{region '#Template'}
	{attribute 'Version' := '0.0.1.0'}
	{attribute 'Tags' := '"LCID": "1031", "Text": "Universal, Analog, Aggregate"'}
	{attribute 'Tags' := '"LCID": "1033", "Text": "Universal, Analog, Aggregate"'}
	{attribute 'Description' := '"LCID": "1031", "Text": "Aktor binär"'}
	{attribute 'Description' := '"LCID": "1033", "Text": "Actuator binary"'}
{endregion}
FUNCTION_BLOCK FB_BA_ActuatorCmd EXTENDS FB_BA_AggregateB
VAR_OUTPUT
	bCmd							: BOOL;
END_VAR
VAR_INPUT CONSTANT
	Cmd						: FB_BA_BO_IO;			
END_VAR

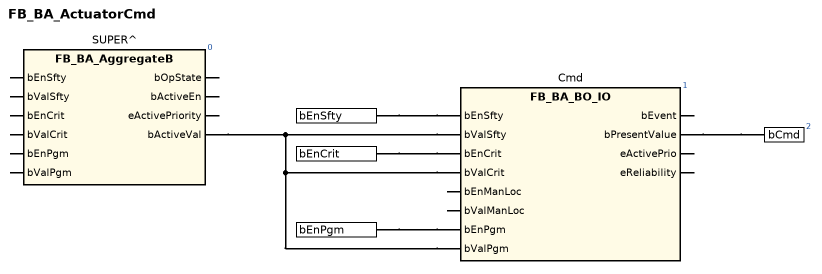
SUPER^(); // FB_BA_AggregateB
Cmd(
    bEnSfty := bEnSfty,
    bValSfty := SUPER^.bActiveVal,
    bEnCrit := bEnCrit,
    bValCrit := SUPER^.bActiveVal,
    bEnPgm := bEnPgm,
    bValPgm := SUPER^.bActiveVal); // FB_BA_BO_IO
bCmd := Cmd.bPresentValue;

METHOD FB_init : BOOL
VAR_INPUT
	bInitRetains : BOOL; // if TRUE, the retain variables are initialized (warm start / cold start)
	bInCopyCode : BOOL;  // if TRUE, the instance afterwards gets moved into the copy code (online change)
END_VAR
Cmd.iParent							:= THIS^;
Cmd.iLabel							:= LblUniFieldDevice.Aggregat_Cmd;			
Cmd.sObjectName						:= '{Idx=01}';	
Cmd.sDeviceType						:= '';
Cmd.bEnOutOfService					:= FALSE;
Cmd.ePolarity						:= E_BA_Polarity.eNormal;
Cmd.eFeedbackPolarity				:= E_BA_Polarity.eNormal;
Cmd.eOverriddenPolarity				:= E_BA_Polarity.eReverse;
Cmd.sActiveText 					:= Texts.txtOn;
Cmd.sInactiveText 					:= Texts.txtOff;
Cmd.nStateChangeCount				:= 0;
Cmd.nActiveTimeElapsed				:= 0;
Cmd.nMinimumOnTime					:= 0;
Cmd.nMinimumOffTime					:= 0;
Cmd.bEnManualRm						:= FALSE;	//	Priority  8	
Cmd.bValManualRm					:= FALSE;	//	Priority  8
Cmd.bDefaultValue					:= FALSE;
Cmd.nEventClassID					:= EventClasses.DisturbanceExtended;
Cmd.stTimeDelay.nToNormal			:= BA2_Param.nDefTimeDelay_ToNormal;
Cmd.stTimeDelay.nToAbnormal			:= BA2_Param.nDefTimeDelay_ToAbnormal;
Cmd.bAcknowledgeRm					:= FALSE;		
Cmd.aEventTransitionText[1]			:= Texts.txtDisturb;
Cmd.aEventTransitionText[2]			:= Texts.txtNone;
Cmd.aEventTransitionText[3]			:= Texts.txtNormal;
Cmd.bEventDetectionEnable			:= FALSE;
Cmd.eEnPlantLock					:= E_BA_LockPriority.eNoLock;
END_METHOD

END_FUNCTION_BLOCK

(* stored: Version 1.1.0.1, ProductVersion 3.1.4024.6
   POU FB_BA_ActuatorCmd: Id {a0af674e-9cdd-4f06-818f-776025190b8d}, SpecialFunc None
   Method FB_init: Id {b90a9b9f-7987-4590-908b-29b6ee3fc5aa} *)
